(* IEC 61131-3 sources: AXOpen/src/integrations/ctrl/src/draft, 3 files *)

(* ---- draft.st ---- *)
NAMESPACE core.draft
    CLASS MainDraft
        VAR PUBLIC
            ixcoreTasks : Tasks;
            ixcoreSequencers : SequencerExample;
        END_VAR

    END_CLASS
END_NAMESPACE

(* ---- ix-core-sequencer.st ---- *)
NAMESPACE core.draft
    using ix.framework.core;

    CLASS SequencerExample EXTENDS ix.framework.core.Context
        VAR PUBLIC
            coord : Sequencer;
        END_VAR

        VAR PUBLIC
            {#ix-set:Description = "Step number one"}
            step_1 : Step;
            {#ix-set:Description = "Step number two"}
            step_2 : Step;
            {#ix-set:Description = "Step number three"}
            step_3 : Step;
            {#ix-set:Description = "Step number four"}
            step_4 : Step;
        END_VAR

        METHOD PROTECTED OVERRIDE Main
            step_1.Initialize(THIS);
            step_2.Initialize(THIS);
            step_3.Initialize(THIS);
            step_4.Initialize(THIS);
            coord.Initialize(THIS);

            coord.Open();

            IF(step_1.Execute(coord)) THEN
                IF((THIS.OpenCycleCount() MOD ULINT#1000) = ULINT#0) THEN
                    coord.MoveNext();
                END_IF;
            END_IF;

            IF(step_2.Execute(coord)) THEN
                IF((THIS.OpenCycleCount() MOD ULINT#1250) = ULINT#0) THEN
                    coord.MoveNext();
                END_IF;
            END_IF;

            IF(step_3.Execute(coord)) THEN
                IF((THIS.OpenCycleCount() MOD ULINT#1500) = ULINT#0) THEN
                    coord.MoveNext();
                END_IF;
            END_IF;
            IF(step_4.Execute(coord)) THEN
                IF((THIS.OpenCycleCount() MOD ULINT#3500) = ULINT#0) THEN
                    coord.MoveNext();
                END_IF;
            END_IF;
        END_METHOD
END_CLASS
END_NAMESPACE

(* ---- ix-core-tasks.st ---- *)
NAMESPACE core.draft
    using ix.framework.core;

    CLASS Tasks EXTENDS ix.framework.core.Context
        VAR PUBLIC
            {#ix-set:AttributeName = "Click to execute this command"}
            _commandTask : CommandTask;
            {#ix-set:AttributeName = "If true the command will end in failure."}
            _commandEndsInFailure : BOOL;
        END_VAR

        VAR a : ULINT; END_VAR
        METHOD PROTECTED OVERRIDE Main
            _commandTask.Initialize(THIS);

            IF(_commandTask.Execute()) THEN
                IF(THIS.OpenCycleCount() MOD ULINT#250 = ULINT#0) THEN
                    if(_commandEndsInFailure) THEN
                        _commandTask.ThrowWhen(TRUE);
                    ELSE
                        _commandTask.DoneWhen(TRUE);
                    END_IF;
                END_IF;
            END_IF;
        END_METHOD
END_CLASS
END_NAMESPACE
